TYPE ST_ENCODER_Status :
STRUCT

	I					: ST_ENCODER_IN;
	Q					: ST_ENCODER_OUT;

END_STRUCT
END_TYPE

(* stored: Version 1.1.0.1
   DUT ST_ENCODER_Status: Id {b77340e5-cb0f-4586-a464-a2dea8e91189} *)
